// SIMATIC S7-200 SMART project (STEP 7-Micro/WIN SMART), CPU ST40

SYMBOL_TABLE Table 1
Start_SW         I0.0
Stop_SW          I0.1
Memory           M0.0
Timer_1          T101
Timer_3          T103
Timer_2          T102
END_SYMBOL_TABLE

ORGANIZATION_BLOCK MAIN:OB1
TITLE=Program Comments
BEGIN
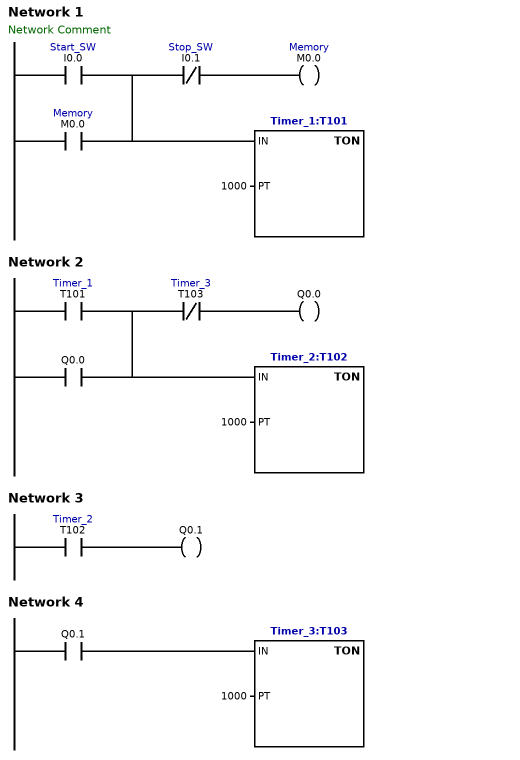
Network 1
// Network Comment
LD     Start_SW:I0.0
O      Memory:M0.0
LPS
AN     Stop_SW:I0.1
=      Memory:M0.0
LPP
TON    Timer_1:T101, 1000
Network 2
LD     Timer_1:T101
O      Q0.0
LPS
AN     Timer_3:T103
=      Q0.0
LPP
TON    Timer_2:T102, 1000
Network 3
LD     Timer_2:T102
=      Q0.1
Network 4
LD     Q0.1
TON    Timer_3:T103, 1000
END_ORGANIZATION_BLOCK
